Fanuc TP program (LS listing): TOOL01_SOUFFLAGE_ON.LS

/PROG  TOOL01_SOUFFLAGE_ON
/ATTR
OWNER		= MNEDITOR;
COMMENT		= "Soufflage ON";
PROG_SIZE	= 132;
CREATE		= DATE 25-04-30  TIME 08:27:30;
MODIFIED	= DATE 25-04-30  TIME 08:27:30;
FILE_NAME	= ;
VERSION		= 0;
LINE_COUNT	= 0;
MEMORY_SIZE	= 376;
PROTECT		= READ_WRITE;
TCD:  STACK_SIZE	= 0,
      TASK_PRIORITY	= 50,
      TIME_SLICE	= 0,
      BUSY_LAMP_OFF	= 0,
      ABORT_REQUEST	= 0,
      PAUSE_REQUEST	= 0;
DEFAULT_GROUP	= 1,*,*,*,*;
CONTROL_CODE	= 00000000 00000000;
/MN
/POS
/END
